INTERFACE I_ArgsBuffer

PROPERTY nArgsLength : UDINT
GET
END_GET
END_PROPERTY

PROPERTY nRetValLength : UDINT
GET
END_GET
END_PROPERTY

PROPERTY pArgsBuffer : POINTER TO BYTE
GET
END_GET
END_PROPERTY

PROPERTY pRetValBuffer : POINTER TO BYTE
GET
END_GET
END_PROPERTY

END_INTERFACE

(* stored: Version 1.1.0.1, ProductVersion 3.1.4024.12
   Itf I_ArgsBuffer: Id {65cdd72b-1ddc-4407-8b79-887e4a3bb4e4}
   Property nArgsLength: Id {f3f09894-ef6d-4f36-b386-c1e57f0d054f}
   Get Get: Id {450d33f4-7513-49de-a50f-85769b95dad8}
   Property nRetValLength: Id {320f8c47-ee1c-4f27-83be-9ada31a05186}
   Get Get: Id {df4b17fa-d390-425c-9bd8-79ce6fbe65ef}
   Property pArgsBuffer: Id {e4bf0197-c4c9-4d06-84c3-2232959f9d61}
   Get Get: Id {6d6fd156-0ec4-4abb-8032-23a6146b2b29}
   Property pRetValBuffer: Id {ce7fe5dc-b9e0-4679-b8f2-34a9f8606a6b}
   Get Get: Id {0c174ef9-ae21-43a1-b164-fd9fa7e2d0f1} *)
